INTERFACE ITF_Axis_Continuous

PROPERTY ModuloFactor : LREAL
GET
END_GET
END_PROPERTY

PROPERTY ModuloPosition : LREAL
GET
END_GET
END_PROPERTY

METHOD SetAxisModuloFactor : BOOL
VAR_INPUT
	fSetAxisModuloFactor		: LREAL;
END_VAR
END_METHOD

END_INTERFACE

(* stored: Version 1.1.0.1, ProductVersion 3.1.4024.9
   Itf ITF_Axis_Continuous: Id {739012a7-325e-40da-9ca5-16dd19a0a1ee}
   Property ModuloFactor: Id {ed37104b-c617-4262-84d6-86fa4b88f2a8}
   Get Get: Id {e35ec7b8-a42d-443f-ae25-fe5f6124f550}
   Property ModuloPosition: Id {101c3772-0a06-4440-a3b7-f721ee9d30c1}
   Get Get: Id {2df4eb48-d0d1-46c7-9713-7362b4127361}
   Method SetAxisModuloFactor: Id {dae37737-eac4-472a-8957-11e0b8617ed4} *)
